Staubli VAL3: ReplyType.pjx

--- ReplyType.pjx ---
Parameters version=s7.3 stackSize=5000 millimeterUnit=true
Data file=ReplyType.dtx

--- ReplyType.dtx ---
public num nSuccess = 1
public num nFailure = 2
